{attribute 'qualified_only'}
VAR_GLOBAL
	P1R AT %Q*: BOOL;	// Zeiger 1 - Rechts
	P1L AT %Q*: BOOL;	// Zeiger 1 - Links
	P2R AT %Q*: BOOL;	// Zeiger 2 - Rechts
	P2L AT %Q*: BOOL;	// Zeiger 2 - Links
	P3R AT %Q*: BOOL;	// Zeiger 3 - Rechts
	P3L AT %Q*: BOOL;	// Zeiger 3 - Links
	P4R AT %Q*: BOOL;	// Zeiger 4 - Rechts
	P4L AT %Q*: BOOL;	// Zeiger 4 - Links
	P5R AT %Q*: BOOL;	// Zeiger 5 - Rechts
	P5L AT %Q*: BOOL;	// Zeiger 5 - Links
END_VAR

(* stored: Version 1.1.0.1, ProductVersion 3.1.4024.4
   GVL SimDA: Id {efa3d63a-96e1-4204-b1e7-9f3703bd4f03} *)
